    // ==============================
    // INTERNAL (optional)
    // ==============================
    aocSpeedTarget              : REAL;      // target line speed during AOC (m/min)
END_VAR

VAR CONSTANT
    // ==============================
    // LIFE CYCLE
    // ==============================
    STATUS_NO_CALL                  : WORD := 16#7000;
    STATUS_FB_FIRST_CALL            : WORD := 16#7001;

    // ==============================
    // AOC STATES
    // ==============================
    STATUS_CHECK_CONDITIONS         : WORD := 16#8000;
    STATUS_SAVE_DF_SPEED            : WORD := 16#8001;
    STATUS_REDUCE_DF_SPEED          : WORD := 16#8002;

    STATUS_ROTARY_SHEAR_CUT_X1      : WORD := 16#8003;
    STATUS_WAIT_ROTARY_SHEAR_CUT_X1 : WORD := 16#8103;

    STATUS_INCREASE_DRYEND_SPEED    : WORD := 16#8004;
    STATUS_CHANGE_SLT_ORDER         : WORD := 16#8005;
    STATUS_CHANGE_RK_SHEET_LENGTH   : WORD := 16#8006;
    STATUS_STK_DISCHARGE            : WORD := 16#8007;

    STATUS_AOC_FINISHED             : WORD := 16#8010;
END_VAR

// =================================================================================================
// CPNTeck - Automação ind.
// (c)Copyright 2022 All Rights Reserved
// -------------------------------------------------------------------------------------------------
// Purpose: Automatic Order Change (AOC) sequence controller.
// Steps (high-level):
//   1) Check material presence
//   2) Reduce double facer speed down to AOC speed
//   3) Execute single cut (rotary shear X1)
//   4) Switch reference to AOC ramp and clear dry-end/slitter
//   5) Update slitter parameters from nextOrder
//   6) Change rotary knife sheet length (delay / clearance window)
//   7) Discharge stacker
//   8) Finish and reset
//
// Notes (important):
// - TP/TON instances are called once per scan at the end of the FB.
// - Requests (reqTp*/reqTon*) are set inside the state machine.
// - This avoids conflicting multi-calls to the same FB instance.
// =================================================================================================


// =================================================================================================
// 1) EDGE HANDLING / DISABLE RESET
// =================================================================================================
rExecuteAOC := executeAOC AND NOT executeAOC_Old;
executeAOC_Old := executeAOC;

// Falling edge of enable => hard reset (safe state)
IF (NOT enable) AND enableOld THEN
    // ---- outputs ----
    error := FALSE;
    aocRunning := FALSE;
    aocTimeOut := FALSE;
    statusDisplay := 'Not running...';

    referenceSwitch := FALSE;
    doubleFacerSpeedUP := FALSE;
    doubleFacerSpeedDown := FALSE;

    rotaryShearCutX1 := FALSE;
    executePositioning := FALSE;
    topStackerDischarge := FALSE;
    bottomStackerDischarge := FALSE;

    rotaryKnifeSpeedRef := 0.0;
    slitterKnifeSpeedRef := 0.0;
    slitterScorerSpeedRef := 0.0;

    // ---- state ----
    stateMachine := STATUS_NO_CALL;

    // ---- reset requests ----
    reqTpRotaryShear := FALSE;
    reqTpExecutePositioning := FALSE;
    reqTpStackerTop := FALSE;
    reqTpStackerBottom := FALSE;

    reqTonSlitterDelay := FALSE;
    reqTonStackerDelay := FALSE;
    reqTonChangeSheetLength := FALSE;

    // ---- stop timeout ----
    tonAocTimeout.IN := FALSE;

    enableOld := enable;
    RETURN;
END_IF

// Rising edge of enable => initialize
IF enable AND (NOT enableOld) THEN
    stateMachine := STATUS_FB_FIRST_CALL;

    // Keep outputs in safe defaults
    error := FALSE;
    aocRunning := FALSE;
    aocTimeOut := FALSE;
    statusDisplay := 'Initialized';

    enableOld := enable;
    RETURN;
END_IF

// If not enabled, do nothing
IF NOT enable THEN
    enableOld := enable;
    RETURN;
END_IF

enableOld := enable;


// =================================================================================================
// 2) DEFAULTS EACH SCAN (avoid latching unwanted outputs)
// =================================================================================================
rotaryShearCutX1 := FALSE;
executePositioning := FALSE;
topStackerDischarge := FALSE;
bottomStackerDischarge := FALSE;

doubleFacerSpeedUP := FALSE;
doubleFacerSpeedDown := FALSE;

// Requests default OFF; states will enable them as needed
reqTpRotaryShear := FALSE;
reqTpExecutePositioning := FALSE;
reqTpStackerTop := FALSE;
reqTpStackerBottom := FALSE;

reqTonSlitterDelay := FALSE;
reqTonStackerDelay := FALSE;
reqTonChangeSheetLength := FALSE;


// =================================================================================================
// 3) TRIGGER AOC (rising edge)
// =================================================================================================
IF rExecuteAOC THEN
    aocTimeOut := FALSE;
    stateMachine := STATUS_CHECK_CONDITIONS;
END_IF


// =================================================================================================
// 4) STATE MACHINE
// =================================================================================================
CASE stateMachine OF

    STATUS_FB_FIRST_CALL:
        statusDisplay := 'FB first call';
        stateMachine := STATUS_NO_CALL;

    STATUS_NO_CALL:
        statusDisplay := 'Idle';
        aocRunning := FALSE;
        referenceSwitch := FALSE;
        tonAocTimeout.IN := FALSE;

    STATUS_CHECK_CONDITIONS:
        statusDisplay := 'Checking conditions';

        // Must have paper present everywhere to proceed
        IF (NOT measuringWheelPaperSensor)
           OR (NOT slitterPaperPresenceSensor)
           OR (NOT rotaryKnifePaperSensor) THEN

            // Not safe to run AOC, finish immediately
            stateMachine := STATUS_AOC_FINISHED;
        ELSE
            // Start timeout supervision
            tonAocTimeout.IN := TRUE;
            tonAocTimeout.PT := configuration.aocTimeout;

            stateMachine := STATUS_SAVE_DF_SPEED;
        END_IF


    STATUS_SAVE_DF_SPEED:
        statusDisplay := 'STATUS_SAVE_DF_SPEED';
        aocRunning := TRUE;

        // Compute AOC target speed (m/min)
        aocSpeedTarget := configuration.automaticOrderChangeSpeed * configuration.automaticOrderChangeSpeedMult;

        stateMachine := STATUS_REDUCE_DF_SPEED;


    STATUS_REDUCE_DF_SPEED:
        statusDisplay := 'STATUS_REDUCE_DF_SPEED';

        // While above AOC speed => pulse DF speed down
        IF lineSpeedMPM > configuration.automaticOrderChangeSpeed THEN
            doubleFacerSpeedDown := instGEN_PULSESpeedCtrl.Q;
        ELSE
            // Reached speed => go cut
            stateMachine := STATUS_ROTARY_SHEAR_CUT_X1;
        END_IF

        // Freeze ramp output to current speed (no AOC ramp yet)
        instFB_Gen_SRamp.X          := lineSpeedMPM;
        instFB_Gen_SRamp.LIMIT_LOW  := lineSpeedMPM;
        instFB_Gen_SRamp.LIMIT_HIGH := lineSpeedMPM;


    STATUS_ROTARY_SHEAR_CUT_X1:
        statusDisplay := 'Cutting web (X1)';
        // Generate a 1s pulse to the shear output
        reqTpRotaryShear := TRUE;
        stateMachine := STATUS_WAIT_ROTARY_SHEAR_CUT_X1;


    STATUS_WAIT_ROTARY_SHEAR_CUT_X1:
        statusDisplay := 'Waiting shear sensor';

        // Wait for confirmation sensor
        IF rotaryShearCutSensor THEN
            // Switch reference to AOC ramp
            referenceSwitch := TRUE;
            stateMachine := STATUS_INCREASE_DRYEND_SPEED;
        END_IF


    STATUS_INCREASE_DRYEND_SPEED:
        statusDisplay := 'Clearing dry-end / slitter';

        // Wait until measuring wheel area clears
        IF NOT measuringWheelPaperSensor THEN
            stateMachine := STATUS_CHANGE_SLT_ORDER;
        END_IF

        // Apply AOC speed ramp (raise limit high to target)
        instFB_Gen_SRamp.X          := aocSpeedTarget;
        instFB_Gen_SRamp.LIMIT_LOW  := lineSpeedMPM;     // don’t ramp below current
        instFB_Gen_SRamp.LIMIT_HIGH := aocSpeedTarget;


    STATUS_CHANGE_SLT_ORDER:
        statusDisplay := 'Changing slitter order (when clear)';

        // Copy only the parameters that need to switch during AOC
        currentOrder.fluteType     := nextOrder.fluteType;
        currentOrder.levelSelector := nextOrder.levelSelector;

        currentOrder.order1.sheetType     := nextOrder.order1.sheetType;
        currentOrder.order1.sheetQuantity := nextOrder.order1.sheetQuantity;
        currentOrder.order1.sheetM1       := nextOrder.order1.sheetM1;
        currentOrder.order1.sheetM2       := nextOrder.order1.sheetM2;
        currentOrder.order1.sheetM3       := nextOrder.order1.sheetM3;
        currentOrder.order1.sheetM4       := nextOrder.order1.sheetM4;
        currentOrder.order1.sheetM5       := nextOrder.order1.sheetM5;

        currentOrder.order2.sheetType     := nextOrder.order2.sheetType;
        currentOrder.order2.sheetQuantity := nextOrder.order2.sheetQuantity;
        currentOrder.order2.sheetM1       := nextOrder.order2.sheetM1;
        currentOrder.order2.sheetM2       := nextOrder.order2.sheetM2;
        currentOrder.order2.sheetM3       := nextOrder.order2.sheetM3;
        currentOrder.order2.sheetM4       := nextOrder.order2.sheetM4;
        currentOrder.order2.sheetM5       := nextOrder.order2.sheetM5;

        // Start delay only after slitter area becomes clear
        IF NOT slitterPaperPresenceSensor THEN
            reqTonSlitterDelay := TRUE;
            tonSlitterPresenceDelay.PT := configuration.slitterPaperPresenceDelay;
        END_IF

        IF tonSlitterPresenceDelay.Q THEN
            // Pulse executePositioning
            reqTpExecutePositioning := TRUE;

            // stop delay timer (will reset by IN=FALSE)
            reqTonSlitterDelay := FALSE;

            stateMachine := STATUS_CHANGE_RK_SHEET_LENGTH;
        END_IF


    STATUS_CHANGE_RK_SHEET_LENGTH:
        statusDisplay := 'Changing rotary knife sheet length';

        // Allow a clearance window for RK sheet length change (time-based + sensor-based)
        reqTonChangeSheetLength := TRUE;
        tonChangeSheetLength.PT := configuration.changeSheetLengthTime;

        // When RK is clear OR timer elapsed => proceed
        IF (NOT rotaryKnifePaperSensor) OR tonChangeSheetLength.Q THEN
            reqTonChangeSheetLength := FALSE;
			currentOrder.changeOrderRequest := TRUE;
            stateMachine := STATUS_STK_DISCHARGE;
        END_IF


    STATUS_STK_DISCHARGE:
        statusDisplay := 'Discharging stacker';

        // Delay before discharge
        reqTonStackerDelay := TRUE;
        tonStackerDischargeDelay.PT := configuration.stackerDischargeDelay;

        IF tonStackerDischargeDelay.Q THEN
            // Pulse discharge commands
            reqTpStackerTop := TRUE;
            reqTpStackerBottom := TRUE;

            // Once pulses are done, finish
            // (TP outputs will be active for PT time; we can finish immediately or wait—here we finish)
            stateMachine := STATUS_AOC_FINISHED;
        END_IF


    STATUS_AOC_FINISHED:
        statusDisplay := 'AOC Finished';

        aocRunning := FALSE;
        referenceSwitch := FALSE;
        doubleFacerSpeedUP := FALSE;
        doubleFacerSpeedDown := FALSE;

        // Stop timeout monitoring
        tonAocTimeout.IN := FALSE;

        // Return to idle
        stateMachine := STATUS_NO_CALL;

END_CASE


// =================================================================================================
// 5) GLOBAL FUNCTION BLOCK CALLS (call once per scan)
// =================================================================================================

// Pulse generator for DF speed up/down buttons
instGEN_PULSESpeedCtrl(
    ENQ := TRUE,
    PTH := configuration.speedControlPulseONTime,
    PTL := configuration.speedControlPulseOFFTime
);

// Ramp block (driven by instFB_Gen_SRamp.X and limits set in states)
instFB_Gen_SRamp(
    A_UP    := configuration.rampUpTimeSec,
    A_DN    := configuration.rampDownTimeSec,
    VU_MAX  := 1000.0,
    VD_MAX  := -1000.0,
    Y       => lineSpeedMPMRamp
);

// Timers
tonSlitterPresenceDelay(IN := reqTonSlitterDelay);
tonStackerDischargeDelay(IN := reqTonStackerDelay);
tonChangeSheetLength(IN := reqTonChangeSheetLength);

tonAocTimeout(IN := tonAocTimeout.IN, PT := configuration.aocTimeout);

// Pulses
tpRotaryShear(IN := reqTpRotaryShear, PT := T#1S, Q => rotaryShearCutX1);
tpExecutePositioning(IN := reqTpExecutePositioning, PT := T#1S, Q => executePositioning);
tpStackerTop(IN := reqTpStackerTop, PT := T#1S, Q => topStackerDischarge);
tpStackerBottom(IN := reqTpStackerBottom, PT := T#1S, Q => bottomStackerDischarge);


// =================================================================================================
// 6) REFERENCES (derived from ramp output)
// =================================================================================================
rotaryKnifeSpeedRef   := lineSpeedMPMRamp * configuration.rotaryKnifeSpeedMult;
slitterKnifeSpeedRef  := lineSpeedMPMRamp * configuration.slitterSpeedMult;
slitterScorerSpeedRef := lineSpeedMPMRamp * configuration.slitterSpeedMult;


// =================================================================================================
// 7) TIMEOUT HANDLING
// =================================================================================================
IF tonAocTimeout.Q THEN
    tonAocTimeout.IN := FALSE;
    aocTimeOut := TRUE;
    stateMachine := STATUS_AOC_FINISHED;
END_IF

END_FUNCTION_BLOCK

// ---- Library/Machine/Rotary knife/Function Block/FB_RotaryKnife_1.TcPOU
FUNCTION_BLOCK FB_RotaryKnife_1




VAR_OUTPUT
    //────────────────────────────────────────────
    // GENERAL / ALARMS (COMMON)
    //────────────────────────────────────────────
    alarmActive                     : BOOL;  // Global alarm active / Alarme geral ativo

    //────────────────────────────────────────────
    // UPPER LEVEL — ENABLE / RUN COMMANDS
    //────────────────────────────────────────────
    upperLevelEnable                : BOOL;  // Upper level enable / Habilita nível superior
    upperLevelInFeedRun             : BOOL;  // Upper infeed run / Partida infeed superior
    upperLevelOutFeedRun            : BOOL;  // Upper outfeed run / Partida outfeed superior
    upperLevelSlave1Run             : BOOL;  // Upper slave1 run / Partida slave1 superior
    upperLevelSlave2Run             : BOOL;  // Upper slave2 run / Partida slave2 superior

    //────────────────────────────────────────────
    // UPPER LEVEL — MOTION / CUT / HOME COMMANDS
    //────────────────────────────────────────────
    upperLevelJogFw                 : BOOL;  // Upper jog forward / JOG avanço superior
    upperLevelJogRev                : BOOL;  // Upper jog reverse / JOG reverso superior
    upperLevelCut                   : BOOL;  // Upper cut command output / Saída corte superior
    upperLevelHome                  : BOOL;  // Upper home command output / Saída home superior
    upperLevelHomeSensorPulse       : BOOL;  // Upper home sensor pulse / Pulso sensor home superior

    //────────────────────────────────────────────
    // UPPER LEVEL — RESET STATUS
    //────────────────────────────────────────────
    upperLevelReset                 : BOOL;  // Upper reset active / Reset superior ativo

    //────────────────────────────────────────────
    // UPPER LEVEL — SPEED REFERENCES
    //────────────────────────────────────────────
    upperLevelInFeedDriveRef        : REAL;  // Upper infeed speed reference / Referência velocidade infeed superior
    upperLevelOutFeedDriveRef       : REAL;  // Upper outfeed speed reference / Referência velocidade outfeed superior

    //────────────────────────────────────────────
    // UPPER LEVEL — ENCODER SELECTION OUTPUT
    //────────────────────────────────────────────
    upperLevelEncoderSwitch         : BOOL;  // Upper encoder select (to drive/IO) / Seletor encoder superior

    //────────────────────────────────────────────
    // LOWER LEVEL — ENABLE / RUN COMMANDS (CREATED)
    //────────────────────────────────────────────
    lowerLevelEnable                : BOOL;  // Lower level enable / Habilita nível inferior
    lowerLevelInFeedRun             : BOOL;  // Lower infeed run / Partida infeed inferior
    lowerLevelOutFeedRun            : BOOL;  // Lower outfeed run / Partida outfeed inferior
    lowerLevelSlave1Run             : BOOL;  // Lower slave1 run / Partida slave1 inferior
    lowerLevelSlave2Run             : BOOL;  // Lower slave2 run / Partida slave2 inferior

    //────────────────────────────────────────────
    // LOWER LEVEL — MOTION / CUT / HOME COMMANDS (CREATED)
    //────────────────────────────────────────────
    lowerLevelJogFw                 : BOOL;  // Lower jog forward / JOG avanço inferior
    lowerLevelJogRev                : BOOL;  // Lower jog reverse / JOG reverso inferior
    lowerLevelCut                   : BOOL;  // Lower cut command output / Saída corte inferior
    lowerLevelHome                  : BOOL;  // Lower home command output / Saída home inferior
    lowerLevelHomeSensorPulse       : BOOL;  // Lower home sensor pulse / Pulso sensor home inferior

    //────────────────────────────────────────────
    // LOWER LEVEL — RESET STATUS (CREATED)
    //────────────────────────────────────────────
    lowerLevelReset                 : BOOL;  // Lower reset active / Reset inferior ativo

    //────────────────────────────────────────────
    // LOWER LEVEL — SPEED REFERENCES (CREATED)
    //────────────────────────────────────────────
    lowerLevelInFeedDriveRef        : REAL;  // Lower infeed speed reference / Referência velocidade infeed inferior
    lowerLevelOutFeedDriveRef       : REAL;  // Lower outfeed speed reference / Referência velocidade outfeed inferior

    //────────────────────────────────────────────
    // LOWER LEVEL — ENCODER SELECTION OUTPUT (CREATED)
    //────────────────────────────────────────────
    lowerLevelEncoderSwitch         : BOOL;  // Lower encoder select (to drive/IO) / Seletor encoder inferior

    //────────────────────────────────────────────
    // HMI STATUS (COMMON)
    //────────────────────────────────────────────
    hmiStatus                       : hmiStatus_TypeStruct; // HMI status structure / Estrutura status HMI
END_VAR
VAR
    //────────────────────────────────────────────
    // UPPER LEVEL — INTERNAL SEQUENCE / STATE
    //────────────────────────────────────────────
    upperLevelStep                 : INT := 0;      // Sequence step for upper level

    //────────────────────────────────────────────
    // UPPER LEVEL — INTERNAL AGGREGATIONS / FLAGS
    //────────────────────────────────────────────
    upperLevelAllDrivesOK          : BOOL := FALSE; // Aggregated drive OK status

    //────────────────────────────────────────────
    // UPPER LEVEL — EDGE DETECTORS
    //────────────────────────────────────────────
    upperLevelRtEnable             : R_TRIG;        // Rising edge for Power ON command
    upperLevelRtPowerOff           : R_TRIG;        // Rising edge for Power OFF command

    //────────────────────────────────────────────
    // UPPER LEVEL — TIMERS
    //────────────────────────────────────────────
    upperLevelTimerReset           : TON;           // 2s reset pulse timer
    upperLevelTimerPulse           : TON;           // General wait/pulse timer used in step 20
    upperLevelTimerWait            : TON;           // Reserved (used in safety reset section)
    upperLevelTimerClear           : TON;           // Reserved (used in safety reset section)

    //────────────────────────────────────────────
    // LOWER LEVEL — INTERNAL SEQUENCE / STATE (CREATED)
    //────────────────────────────────────────────
    lowerLevelStep                 : INT := 0;      // Sequence step for lower level

    //────────────────────────────────────────────
    // LOWER LEVEL — INTERNAL AGGREGATIONS / FLAGS (CREATED)
    //────────────────────────────────────────────
    lowerLevelAllDrivesOK          : BOOL := FALSE; // Aggregated drive OK status

    //────────────────────────────────────────────
    // LOWER LEVEL — EDGE DETECTORS (CREATED)
    //────────────────────────────────────────────
    lowerLevelRtEnable             : R_TRIG;        // Rising edge for Power ON command
    lowerLevelRtPowerOff           : R_TRIG;        // Rising edge for Power OFF command

    //────────────────────────────────────────────
    // LOWER LEVEL — TIMERS (CREATED)
    //────────────────────────────────────────────
    lowerLevelTimerReset           : TON;           // 2s reset pulse timer
    lowerLevelTimerPulse           : TON;           // General wait/pulse timer used in step 20
    lowerLevelTimerWait            : TON;           // Reserved (used in safety reset section)
    lowerLevelTimerClear           : TON;           // Reserved (used in safety reset section)

    //────────────────────────────────────────────
    // MODBUS TCP — FUNCTION BLOCKS / GLOBAL STATE
    //────────────────────────────────────────────
    instFB_MBReadRegs              : FB_MBReadRegs;   // Modbus TCP read registers FB
    instFB_MBWriteRegs             : FB_MBWriteRegs;  // Modbus TCP write registers FB
    modbusTCPStep                  : INT;             // Modbus TCP state machine step

    //────────────────────────────────────────────
    // MODBUS TCP — UPPER LEVEL DATA
    //────────────────────────────────────────────
    upperLevelStatusWord1          : INT;
    upperLevelStatusWord2          : INT;
    upperLevelModbusDword          : DWORD;
    upperLevelWriteMenu2029        : DWORD;
    upperLevelLineSpeed            : WORD;
	upperLevelStatusW1				: rotaryKnifeStatusWord1_TypeStruct;
	upperLevelStatusW2				: rotaryKnifeStatusWord2_TypeStruct;		

    //────────────────────────────────────────────
    // MODBUS TCP — LOWER LEVEL DATA
    //────────────────────────────────────────────
    lowerLevelStatusWord1          : INT;
    lowerLevelStatusWord2          : INT;
    lowerLevelModbusDword          : DWORD;
    lowerLevelWriteMenu2029        : DWORD;
    lowerLevelLineSpeed            : WORD;

	lowerLevelStatusW1				: rotaryKnifeStatusWord1_TypeStruct;
	lowerLevelStatusW2				: rotaryKnifeStatusWord2_TypeStruct;	
	
	
END_VAR

VAR PERSISTENT
	
	lowerLevelTotalOfCutsAccumulator : DINT;
	upperLevelTotalOfCutsAccumulator : DINT;


END_VAR

VAR_IN_OUT

	currentOrder	: Order_TypeStruct;

END_VAR

_00_ModbusTCP();
_01_UpperLevelControl();
_02_LowerLevelControl();

METHOD _00_ModbusTCP
VAR_INPUT
END_VAR
CASE modbusTCPStep OF
	
		(*________________________________________________________________*)
		00:(*Read lower level line speed*)
	
		instFB_MBReadRegs(
		sIPAddr:= '192.168.100.11', 
		nTCPPort:= 502, 
		nUnitID:= 1, 
		nQuantity:= 1, 
		nMBAddr:= 16#711, (*Menu 18.10*)
		cbLength:= SIZEOF(lowerLevelLineSpeed),  
		pDestAddr:= ADR(lowerLevelLineSpeed),  
		bExecute:= TRUE, 
		tTimeout:= T#500MS,  
		bBusy=> , 
		bError=> , 
		nErrId=> , 
		cbRead=> );
		
	
		IF NOT instFB_MBReadRegs.bBusy THEN
			instFB_MBReadRegs(bExecute:=FALSE);
			modbusTCPStep:=modbusTCPStep + 1;	(*Index*)
		END_IF
		
		
		(*________________________________________________________________*)		
		01:(*Read rotary knife status word1*)
	
		instFB_MBReadRegs(
		sIPAddr:= '192.168.100.11', 
		nTCPPort:= 502, 
		nUnitID:= 1, 
		nQuantity:= 1, 
		nMBAddr:= 16#774, //Parameter #19.09 - 1 = > HEX
		cbLength:= SIZEOF(upperLevelStatusWord1),  
		pDestAddr:= ADR(upperLevelStatusWord1),  
		bExecute:= TRUE,  
		tTimeout:= T#500MS,  
		bBusy=> , 
		bError=> , 
		nErrId=> , 
		cbRead=> );
		
		IF NOT instFB_MBReadRegs.bBusy THEN
			instFB_MBReadRegs(bExecute:=FALSE);
			modbusTCPStep:=modbusTCPStep + 1;	(*Index*)			
		END_IF	
		
		
		(*________________________________________________________________*)		
		02:(*Read rotary knife status word1*)
	
		instFB_MBReadRegs(
		sIPAddr:= '192.168.100.11', 
		nTCPPort:= 502, 
		nUnitID:= 1, 
		nQuantity:= 1, 
		nMBAddr:= 16#775, //Parameter #19.10 - 1 = > HEX
		cbLength:= SIZEOF(upperLevelStatusWord2),  
		pDestAddr:= ADR(upperLevelStatusWord2),  
		bExecute:= TRUE,  
		tTimeout:= T#500MS,  
		bBusy=> , 
		bError=> , 
		nErrId=> , 
		cbRead=> );
		
		IF NOT instFB_MBReadRegs.bBusy THEN
			instFB_MBReadRegs(bExecute:=FALSE);
			modbusTCPStep:=modbusTCPStep + 1;	(*Index*)

		END_IF			





		(*________________________________________________________________*)
		03:(*Read lower level line speed*)
	
		instFB_MBReadRegs(
		sIPAddr:= '192.168.100.12', 
		nTCPPort:= 502, 
		nUnitID:= 1, 
		nQuantity:= 1, 
		nMBAddr:= 16#711, (*Menu 18.10*)
		cbLength:= SIZEOF(lowerLevelLineSpeed),  
		pDestAddr:= ADR(lowerLevelLineSpeed),  
		bExecute:= TRUE, 
		tTimeout:= T#500MS,  
		bBusy=> , 
		bError=> , 
		nErrId=> , 
		cbRead=> );
		
	
		IF NOT instFB_MBReadRegs.bBusy THEN
			instFB_MBReadRegs(bExecute:=FALSE);
			modbusTCPStep:=modbusTCPStep + 1;	(*Index*)
		END_IF
		
		
		(*________________________________________________________________*)		
		04:(*Read rotary knife status word1*)
	
		instFB_MBReadRegs(
		sIPAddr:= '192.168.100.12', 
		nTCPPort:= 502, 
		nUnitID:= 1, 
		nQuantity:= 1, 
		nMBAddr:= 16#774, //Parameter #19.09 - 1 = > HEX
		cbLength:= SIZEOF(lowerLevelStatusWord1),  
		pDestAddr:= ADR(lowerLevelStatusWord1),  
		bExecute:= TRUE,  
		tTimeout:= T#500MS,  
		bBusy=> , 
		bError=> , 
		nErrId=> , 
		cbRead=> );
		
		
		IF NOT instFB_MBReadRegs.bBusy THEN
			instFB_MBReadRegs(bExecute:=FALSE);
			modbusTCPStep:=modbusTCPStep + 1;	(*Index*)			
		END_IF	
		
		(*________________________________________________________________*)		
		05:(*Read rotary knife status word1*)
	
		instFB_MBReadRegs(
		sIPAddr:= '192.168.100.12', 
		nTCPPort:= 502, 
		nUnitID:= 1, 
		nQuantity:= 1, 
		nMBAddr:= 16#775, //Parameter #19.10 - 1 = > HEX
		cbLength:= SIZEOF(lowerLevelStatusWord2),  
		pDestAddr:= ADR(lowerLevelStatusWord2),  
		bExecute:= TRUE,  
		tTimeout:= T#500MS,  
		bBusy=> , 
		bError=> , 
		nErrId=> , 
		cbRead=> );
		
		IF NOT instFB_MBReadRegs.bBusy THEN
			instFB_MBReadRegs(bExecute:=FALSE);
			modbusTCPStep:=modbusTCPStep + 1;	(*Index*)

		END_IF	
		
		
		
	(*________________________________________________________________*)	
		6:(*Write lower level sheet lenght*)	
	
		
		IF NOT currentOrder.invertOrderLevel THEN
			
			upperLevelModbusDword := (INT_TO_DWORD(currentOrder.order1.sheetLength) * 1000);
	
		ELSE
			
			upperLevelModbusDword := (INT_TO_DWORD(currentOrder.order2.sheetLength) * 1000);			
		
		END_IF
					
		upperLevelWriteMenu2029 := SHR(upperLevelModbusDword,16) OR SHL(upperLevelModbusDword,16);
		
		//Write menu 20.29 - MBAddres: 16#47EC (18412dec)
		instFB_MBWriteRegs(
		sIPAddr:= '192.168.100.11', //Modbus gateway IP Addres
		nTCPPort:= 502, //Modbus gateway port
		nUnitID:= 1, //Drive addres subnode
		nQuantity:= 2, //Number of words
		nMBAddr:= 16#47EC, 
		cbLength:= SIZEOF(upperLevelWriteMenu2029), 
		pSrcAddr:= ADR(upperLevelWriteMenu2029), 
		bExecute:= TRUE, 
		tTimeout:= T#1000MS, 
		bBusy=> , 
		bError=> , 
		nErrId=> );
		
		IF NOT instFB_MBWriteRegs.bBusy THEN
			instFB_MBWriteRegs(bExecute:=FALSE);
			modbusTCPStep:=modbusTCPStep + 1;	(*Index*)

		END_IF			

		
		
		7:(*Write lower level sheet lenght*)	
	
		
		IF NOT currentOrder.invertOrderLevel THEN
			
			lowerLevelModbusDword := (INT_TO_DWORD(currentOrder.order2.sheetLength) * 1000);
	
		ELSE
			
			lowerLevelModbusDword := (INT_TO_DWORD(currentOrder.order1.sheetLength) * 1000);			
		
		END_IF
					
		lowerLevelWriteMenu2029 := SHR(lowerLevelModbusDword,16) OR SHL(lowerLevelModbusDword,16);
		
		//Write menu 20.29 - MBAddres: 16#47EC (18412dec)
		instFB_MBWriteRegs(
		sIPAddr:= '192.168.100.12', //Modbus gateway IP Addres
		nTCPPort:= 502, //Modbus gateway port
		nUnitID:= 1, //Drive addres subnode
		nQuantity:= 2, //Number of words
		nMBAddr:= 16#47EC, 
		cbLength:= SIZEOF(lowerLevelWriteMenu2029), 
		pSrcAddr:= ADR(lowerLevelWriteMenu2029), 
		bExecute:= TRUE, 
		tTimeout:= T#1000MS, 
		bBusy=> , 
		bError=> , 
		nErrId=> );
		
		IF NOT instFB_MBWriteRegs.bBusy THEN
			instFB_MBWriteRegs(bExecute:=FALSE);
			modbusTCPStep:=0;	(*Index*)

		END_IF				
	
END_CASE		



//==============================================================
// STATUS WORD 1 — BIT TO BOOL MAPPING (Upper + Lower)
//==============================================================

//-----------------------------
// Upper Level — Status Word 1
//-----------------------------
upperLevelStatusW1.knifeAtHomeParkPos1              := upperLevelStatusWord1.00;
upperLevelStatusW1.homingInProgress                 := upperLevelStatusWord1.01;
upperLevelStatusW1.homingComplete                   := upperLevelStatusWord1.02;
upperLevelStatusW1.knifeInspectionMotionInProgress  := upperLevelStatusWord1.03;
upperLevelStatusW1.knifeInspectionMotionComplete    := upperLevelStatusWord1.04;
upperLevelStatusW1.returnHomeMotionInProgress       := upperLevelStatusWord1.05;
upperLevelStatusW1.returnHomeMotionComplete         := upperLevelStatusWord1.06;
upperLevelStatusW1.jogForwardInProgress             := upperLevelStatusWord1.07;
upperLevelStatusW1.jogReverseInProgress             := upperLevelStatusWord1.08;
upperLevelStatusW1.knifeGearingOut                  := upperLevelStatusWord1.09;
upperLevelStatusW1.knifeRunningEngaged              := upperLevelStatusWord1.10;
upperLevelStatusW1.knifeStoppedDisengaged           := upperLevelStatusWord1.11;
upperLevelStatusW1.maxLineSpeedLimitCalculated      := upperLevelStatusWord1.12;
upperLevelStatusW1.batchMaxLineSpeedCalcInProgress  := upperLevelStatusWord1.13;
upperLevelStatusW1.batchMaxLineSpeedCalculated      := upperLevelStatusWord1.14;
upperLevelStatusW1.watchdogClockOut                 := upperLevelStatusWord1.15;

//-----------------------------
// Lower Level — Status Word 1
//-----------------------------
lowerLevelStatusW1.knifeAtHomeParkPos1              := lowerLevelStatusWord1.00;
lowerLevelStatusW1.homingInProgress                 := lowerLevelStatusWord1.01;
lowerLevelStatusW1.homingComplete                   := lowerLevelStatusWord1.02;
lowerLevelStatusW1.knifeInspectionMotionInProgress  := lowerLevelStatusWord1.03;
lowerLevelStatusW1.knifeInspectionMotionComplete    := lowerLevelStatusWord1.04;
lowerLevelStatusW1.returnHomeMotionInProgress       := lowerLevelStatusWord1.05;
lowerLevelStatusW1.returnHomeMotionComplete         := lowerLevelStatusWord1.06;
lowerLevelStatusW1.jogForwardInProgress             := lowerLevelStatusWord1.07;
lowerLevelStatusW1.jogReverseInProgress             := lowerLevelStatusWord1.08;
lowerLevelStatusW1.knifeGearingOut                  := lowerLevelStatusWord1.09;
lowerLevelStatusW1.knifeRunningEngaged              := lowerLevelStatusWord1.10;
lowerLevelStatusW1.knifeStoppedDisengaged           := lowerLevelStatusWord1.11;
lowerLevelStatusW1.maxLineSpeedLimitCalculated      := lowerLevelStatusWord1.12;
lowerLevelStatusW1.batchMaxLineSpeedCalcInProgress  := lowerLevelStatusWord1.13;
lowerLevelStatusW1.batchMaxLineSpeedCalculated      := lowerLevelStatusWord1.14;
lowerLevelStatusW1.watchdogClockOut                 := lowerLevelStatusWord1.15;

//==============================================================
// STATUS WORD 2 — BIT TO BOOL MAPPING (Upper + Lower)
//==============================================================

//-----------------------------
// Upper Level — Status Word 2
//-----------------------------
upperLevelStatusW2.batchSingleShotStopInProgress := upperLevelStatusWord2.00;
upperLevelStatusW2.registrationMarkMissed        := upperLevelStatusWord2.01;
upperLevelStatusW2.registrationWindowOpen        := upperLevelStatusWord2.02;
upperLevelStatusW2.registrationMarkAccepted      := upperLevelStatusWord2.03;
upperLevelStatusW2.onLastBatch                   := upperLevelStatusWord2.04;
upperLevelStatusW2.onLastCutOfLastBatch          := upperLevelStatusWord2.05;
upperLevelStatusW2.pls1Output                    := upperLevelStatusWord2.06;
upperLevelStatusW2.pls2Output                    := upperLevelStatusWord2.07;
upperLevelStatusW2.referenceEnabled              := upperLevelStatusWord2.08;
upperLevelStatusW2.driveHealthy                  := upperLevelStatusWord2.09;
upperLevelStatusW2.reserved10                    := upperLevelStatusWord2.10;
upperLevelStatusW2.reserved11                    := upperLevelStatusWord2.11;
upperLevelStatusW2.userDefinedStatusBit12        := upperLevelStatusWord2.12;
upperLevelStatusW2.userDefinedStatusBit13        := upperLevelStatusWord2.13;
upperLevelStatusW2.userDefinedStatusBit14        := upperLevelStatusWord2.14;
upperLevelStatusW2.userDefinedStatusBit15        := upperLevelStatusWord2.15;

//-----------------------------
// Lower Level — Status Word 2
//-----------------------------
lowerLevelStatusW2.batchSingleShotStopInProgress := lowerLevelStatusWord2.00;
lowerLevelStatusW2.registrationMarkMissed        := lowerLevelStatusWord2.01;
lowerLevelStatusW2.registrationWindowOpen        := lowerLevelStatusWord2.02;
lowerLevelStatusW2.registrationMarkAccepted      := lowerLevelStatusWord2.03;
lowerLevelStatusW2.onLastBatch                   := lowerLevelStatusWord2.04;
lowerLevelStatusW2.onLastCutOfLastBatch          := lowerLevelStatusWord2.05;
lowerLevelStatusW2.pls1Output                    := lowerLevelStatusWord2.06;
lowerLevelStatusW2.pls2Output                    := lowerLevelStatusWord2.07;
lowerLevelStatusW2.referenceEnabled              := lowerLevelStatusWord2.08;
lowerLevelStatusW2.driveHealthy                  := lowerLevelStatusWord2.09;
lowerLevelStatusW2.reserved10                    := lowerLevelStatusWord2.10;
lowerLevelStatusW2.reserved11                    := lowerLevelStatusWord2.11;
lowerLevelStatusW2.userDefinedStatusBit12        := lowerLevelStatusWord2.12;
lowerLevelStatusW2.userDefinedStatusBit13        := lowerLevelStatusWord2.13;
lowerLevelStatusW2.userDefinedStatusBit14        := lowerLevelStatusWord2.14;
lowerLevelStatusW2.userDefinedStatusBit15        := lowerLevelStatusWord2.15;
END_METHOD

METHOD _01_UpperLevelControl
VAR_INPUT
END_VAR
(*
======================================================================
UPPER LEVEL — Rotary Knife Control (Upper Knife)
======================================================================
Concept:
- Power ON command starts a simple sequence:
  0  = OFF / Idle
  10 = Enable drives + follow line speed
  20 = Send HOME command for 1s
  21 = Wait for HomingComplete status before running infeed/outfeed
  40 = Normal operation (cut enabled when command + paper present)

Rule:
- When the upper level is powered ON, infeed/outfeed speed references
  must follow lineSpeedMPM.
======================================================================
*)

//==============================================================
// 1) RESET PULSE (2s) + EDGE DETECTION
//==============================================================
upperLevelTimerReset(IN := resetCmd, PT := T#2S);
upperLevelReset := upperLevelTimerReset.Q;

upperLevelRtEnable(CLK := upperLevelPowerONCmd);
upperLevelRtPowerOff(CLK := upperLevelPowerOFFCmd);

//==============================================================
// 2) DRIVE/SAFETY STATUS (AGGREGATION)
//==============================================================
upperLevelAllDrivesOK := upperLevelInfeedDrvOK  AND
                         upperLevelOutfeedDrvOK AND
                         upperLevelMainDrvOK    AND
                         upperLevelSlave1DrvOK  AND
                         upperLevelSlave2DrvOK;

upperLevelHomeSensorPulse := upperLevelHomeSensor;

//==============================================================
// 3) START SEQUENCE CONDITION
//==============================================================
// Start only if:
// - Rising edge on Power ON
// - Sequence is idle
// - Safety chain OK
// - All drives OK
// - No reset pulse active
IF upperLevelRtEnable.Q
   AND (upperLevelStep = 0)
   AND safetyFeedback
   AND upperLevelAllDrivesOK
   AND NOT upperLevelReset THEN

    upperLevelStep := 10;
END_IF

//==============================================================
// 4) SEQUENCE STATE MACHINE
//==============================================================
CASE upperLevelStep OF

    //==========================================================
    // 0 — OFF / IDLE
    //==========================================================
    0:
        // Commands OFF
        upperLevelEnable      := FALSE;
        upperLevelSlave1Run   := FALSE;
        upperLevelSlave2Run   := FALSE;
        upperLevelInFeedRun   := FALSE;
        upperLevelOutFeedRun  := FALSE;

        // Motion / actions OFF
        upperLevelJogFw       := FALSE;
        upperLevelJogRev      := FALSE;
        upperLevelHome        := FALSE;
        upperLevelCut         := FALSE;

        // References = 0
        upperLevelInFeedDriveRef  := 0.0;
        upperLevelOutFeedDriveRef := 0.0;

    //==========================================================
    // 10 — ENABLE DRIVES + FOLLOW LINE SPEED
    //==========================================================
    10:
        upperLevelEnable      := TRUE;
        upperLevelSlave1Run   := TRUE;
        upperLevelSlave2Run   := TRUE;

        // Follow line speed immediately when powered ON
        upperLevelInFeedDriveRef  := lineSpeedMPM;
        upperLevelOutFeedDriveRef := lineSpeedMPM;

        // Next step: issue homing pulse
        upperLevelStep := 20;

    //==========================================================
    // 20 — HOME COMMAND PULSE (1s)
    //==========================================================
    20:
        // Command home for 1 second
        upperLevelHome := TRUE;

        upperLevelTimerPulse(IN := TRUE, PT := T#1S);
        IF upperLevelTimerPulse.Q THEN
            upperLevelHome := FALSE;
            upperLevelTimerPulse(IN := FALSE);
            upperLevelStep := 21;
        END_IF

    //==========================================================
    // 21 — WAIT HOMING COMPLETE
    //==========================================================
    21:

        // Start infeed/outfeed only after homing is complete
        IF upperLevelStatusW1.homingComplete THEN
            upperLevelInFeedRun  := TRUE;
            upperLevelOutFeedRun := TRUE;
            upperLevelStep := 40;
        END_IF

    //==========================================================
    // 40 — NORMAL OPERATION
    //==========================================================
    40:
        // Track line speed continuously
        upperLevelInFeedDriveRef  := lineSpeedMPM;
        upperLevelOutFeedDriveRef := lineSpeedMPM;

        // Enable cut only when commanded and paper present
        upperLevelCut := (upperLevelCutCmd AND upperLevelPaperSensor);

END_CASE

//==============================================================
// 5) GLOBAL INTERLOCK — IMMEDIATE STOP
//==============================================================
// Immediate stop on any of these conditions:
// - Safety chain not OK
// - Any drive not OK
// - Power OFF command rising edge
IF (NOT safetyFeedback) OR (NOT upperLevelAllDrivesOK) OR upperLevelRtPowerOff.Q THEN

    upperLevelStep := 0;

    upperLevelEnable      := FALSE;
    upperLevelSlave1Run   := FALSE;
    upperLevelSlave2Run   := FALSE;
    upperLevelInFeedRun   := FALSE;
    upperLevelOutFeedRun  := FALSE;

    upperLevelJogFw       := FALSE;
    upperLevelJogRev      := FALSE;
    upperLevelHome        := FALSE;
    upperLevelCut         := FALSE;

    upperLevelInFeedDriveRef  := 0.0;
    upperLevelOutFeedDriveRef := 0.0;

    // Reset internal timers for a clean restart
    upperLevelTimerWait(IN := FALSE);
    upperLevelTimerPulse(IN := FALSE);
    upperLevelTimerClear(IN := FALSE);
    upperLevelTimerReset(IN := FALSE);
END_IF
END_METHOD

METHOD _02_LowerLevelControl
VAR_INPUT
END_VAR
(*
======================================================================
LOWER LEVEL — Rotary Knife Control (Lower Knife)
======================================================================
Concept:
- Power ON command starts a simple sequence:
  0  = OFF / Idle
  10 = Enable drives + follow line speed
  20 = Send HOME command for 1s
  21 = Wait for HomingComplete status before running infeed/outfeed
  40 = Normal operation (cut enabled when command + paper present)

Rule:
- When the lower level is powered ON, infeed/outfeed speed references
  must follow lineSpeedMPM.
======================================================================
*)

//==============================================================
// 1) RESET PULSE (2s) + EDGE DETECTION
//==============================================================
lowerLevelTimerReset(IN := resetCmd, PT := T#2S);
lowerLevelReset := lowerLevelTimerReset.Q;

lowerLevelRtEnable(CLK := lowerLevelPowerONCmd);
lowerLevelRtPowerOff(CLK := lowerLevelPowerOFFCmd);

//==============================================================
// 2) DRIVE/SAFETY STATUS (AGGREGATION)
//==============================================================
lowerLevelAllDrivesOK := lowerLevelInfeedDrvOK  AND
                         lowerLevelOutfeedDrvOK AND
                         lowerLevelMainDrvOK    AND
                         lowerLevelSlave1DrvOK  AND
                         lowerLevelSlave2DrvOK;

lowerLevelHomeSensorPulse := lowerLevelHomeSensor;

//==============================================================
// 3) START SEQUENCE CONDITION
//==============================================================
// Start only if:
// - Rising edge on Power ON
// - Sequence is idle
// - Safety chain OK
// - All drives OK
// - No reset pulse active
IF lowerLevelRtEnable.Q
   AND (lowerLevelStep = 0)
   AND safetyFeedback
   AND lowerLevelAllDrivesOK
   AND NOT lowerLevelReset THEN

    lowerLevelStep := 10;
END_IF

//==============================================================
// 4) SEQUENCE STATE MACHINE
//==============================================================
CASE lowerLevelStep OF

    //==========================================================
    // 0 — OFF / IDLE
    //==========================================================
    0:
        // Commands OFF
        lowerLevelEnable      := FALSE;
        lowerLevelSlave1Run   := FALSE;
        lowerLevelSlave2Run   := FALSE;
        lowerLevelInFeedRun   := FALSE;
        lowerLevelOutFeedRun  := FALSE;

        // Motion / actions OFF
        lowerLevelJogFw       := FALSE;
        lowerLevelJogRev      := FALSE;
        lowerLevelHome        := FALSE;
        lowerLevelCut         := FALSE;

        // References = 0
        lowerLevelInFeedDriveRef  := 0.0;
        lowerLevelOutFeedDriveRef := 0.0;

    //==========================================================
    // 10 — ENABLE DRIVES + FOLLOW LINE SPEED
    //==========================================================
    10:
        lowerLevelEnable      := TRUE;
        lowerLevelSlave1Run   := TRUE;
        lowerLevelSlave2Run   := TRUE;

        // Follow line speed immediately when powered ON
        lowerLevelInFeedDriveRef  := lineSpeedMPM;
        lowerLevelOutFeedDriveRef := lineSpeedMPM;

        // Next step: issue homing pulse
        lowerLevelStep := 20;

    //==========================================================
    // 20 — HOME COMMAND PULSE (1s)
    //==========================================================
    20:
        // Command home for 1 second
        lowerLevelHome := TRUE;

        lowerLevelTimerPulse(IN := TRUE, PT := T#1S);
        IF lowerLevelTimerPulse.Q THEN
            lowerLevelHome := FALSE;
            lowerLevelTimerPulse(IN := FALSE);
            lowerLevelStep := 21;
        END_IF

    //==========================================================
    // 21 — WAIT HOMING COMPLETE
    //==========================================================
    21:
        // Start infeed/outfeed only after homing is complete
        IF lowerLevelStatusW1.homingComplete THEN
            lowerLevelInFeedRun  := TRUE;
            lowerLevelOutFeedRun := TRUE;
            lowerLevelStep := 40;
        END_IF

    //==========================================================
    // 40 — NORMAL OPERATION
    //==========================================================
    40:
        // Track line speed continuously
        lowerLevelInFeedDriveRef  := lineSpeedMPM;
        lowerLevelOutFeedDriveRef := lineSpeedMPM;

        // Enable cut only when commanded and paper present
        lowerLevelCut := (lowerLevelCutCmd AND lowerLevelPaperSensor);

END_CASE

//==============================================================
// 5) GLOBAL INTERLOCK — IMMEDIATE STOP
//==============================================================
// Immediate stop on any of these conditions:
// - Safety chain not OK
// - Any drive not OK
// - Power OFF command rising edge
IF (NOT safetyFeedback) OR (NOT lowerLevelAllDrivesOK) OR lowerLevelRtPowerOff.Q THEN

    lowerLevelStep := 0;

    lowerLevelEnable      := FALSE;
    lowerLevelSlave1Run   := FALSE;
    lowerLevelSlave2Run   := FALSE;
    lowerLevelInFeedRun   := FALSE;
    lowerLevelOutFeedRun  := FALSE;

    lowerLevelJogFw       := FALSE;
    lowerLevelJogRev      := FALSE;
    lowerLevelHome        := FALSE;
    lowerLevelCut         := FALSE;

    lowerLevelInFeedDriveRef  := 0.0;
    lowerLevelOutFeedDriveRef := 0.0;

    // Reset internal timers for a clean restart
    lowerLevelTimerWait(IN := FALSE);
    lowerLevelTimerPulse(IN := FALSE);
    lowerLevelTimerClear(IN := FALSE);
    lowerLevelTimerReset(IN := FALSE);
END_IF
END_METHOD

END_FUNCTION_BLOCK

// ---- Library/Machine/Slitter/FunctionBlocks/FB_PaperDirectionControl_.TcPOU
FUNCTION_BLOCK FB_PaperDirectionControl_
VAR_INPUT
	
	executeCmd	: BOOL;
	allUPCmd : BOOL;
	allDownCmd : BOOL;
	invertDirection	: BOOL;
	numberOfFlaps				: INT := 27;
	flapsManualCmdArr			: ARRAY [1..27] OF hmiCommandsFlaps_TypeStruct;	
	currentOrder				: Order_TypeStruct;
	machineConfig				: slitterConfig_TypeStruct; // Slitter configuration parameters / Parâmetros do slitter

END_VAR
VAR_OUTPUT
	
	flapSolenoidArr			: ARRAY [1..27] OF BOOL;	

END_VAR


VAR
	invertDirectionOld	: BOOL;
	executeCmdOld: BOOL;
	i: INT;
END_VAR

// Trigger logic on rising edge of execute command
IF executeCmd AND NOT executeCmdOld THEN

    FOR i := 1 TO numberOfFlaps DO
        
        // 1. Level 1 Only (Upper)
        IF currentOrder.levelSelector = E_LevelSelector.eUpperOnly THEN
            flapSolenoidArr[i] := TRUE;

        // 2. Level 2 Only (Lower)
        ELSIF currentOrder.levelSelector = E_LevelSelector.eLowerOnly THEN
            flapSolenoidArr[i] := FALSE;

        // 3. Both Levels (Decision based on Order 1 Width vs Flap physical position)
        ELSIF currentOrder.levelSelector = E_LevelSelector.eBoth THEN
            
            // If flap is within the width of Order 1, it follows Order 1 direction
            IF machineConfig.arrFlapPosition[i] <= (currentOrder.generatedOrder.order1Width + currentOrder.generatedOrder.firstKnifePosition) THEN
                flapSolenoidArr[i] :=  FALSE;
            ELSE
                // Otherwise it follows Order 2 direction
                flapSolenoidArr[i] :=  TRUE;
            END_IF;

        END_IF;
    END_FOR;

END_IF;
// Update edge detection memory
executeCmdOld := executeCmd;

// Global Overrides (Master Up / Master Down)
// These run regardless of the executeCmd rising edge if triggered
IF allUPCmd THEN
    FOR i := 1 TO 27 DO flapSolenoidArr[i] := TRUE; END_FOR;
ELSIF allDownCmd THEN
    FOR i := 1 TO 27 DO flapSolenoidArr[i] := FALSE; END_FOR;
	
END_IF;

// Manual HMI Control Override (If enabled in the HMI command structure)
FOR i := 1 TO 27 DO
    IF flapsManualCmdArr[i].upCmd THEN
        flapSolenoidArr[i] := TRUE;
    END_IF;
	
    IF flapsManualCmdArr[i].downCmd THEN
        flapSolenoidArr[i] := FALSE;
    END_IF;	
	
END_FOR;

//Invert flap direction
IF invertDirection AND NOT invertDirectionOld THEN
	
	// Loop through all flaps and flip their current solenoid state
	FOR i := 1 TO numberOfFlaps DO
		flapSolenoidArr[i] := NOT flapSolenoidArr[i];
	END_FOR;

END_IF
invertDirectionOld := invertDirection;

END_FUNCTION_BLOCK

// ---- Library/Machine/Slitter/FunctionBlocks/FB_SpeedMeter.TcPOU
FUNCTION_BLOCK FB_SpeedMeter
VAR_INPUT

	mesuringWheelPulseSensor		: BOOL;
	measuringWheelDiameter		: REAL	:= 159.0;
	cycleTimeSeconds			: TIME	:= T#1S;

END_VAR
VAR_OUTPUT

	mesuringWheelSpeedRPM		: REAL;
	measuringWheelSpeedMPM		: REAL;

END_VAR
VAR

	measuringWheelPulseCounter	: DINT;
	measuringWheelPulseCounterOld	: DINT;
	measuringWheelPulseDif		: DINT;
	cycleCounter				: DINT;

	mesuringWheelPulseSensorOld	: BOOL;
	timerPulse					: BOOL;
	timerPulseOld				: BOOL;
	instTimerTON				: TON;

	cycleTimeSecondsInt: INT;
END_VAR



VAR CONSTANT

	PI						: REAL	:= 3.14159265359;

END_VAR



IF mesuringWheelPulseSensor AND NOT mesuringWheelPulseSensorOld THEN

	measuringWheelPulseCounter := measuringWheelPulseCounter + 1;

END_IF

mesuringWheelPulseSensorOld := mesuringWheelPulseSensor;




IF instTimerTON.Q THEN

	timerPulse := FALSE;
	instTimerTON.IN	:= FALSE;

END_IF

IF NOT instTimerTON.IN AND NOT instTimerTON.Q THEN

	timerPulse := TRUE;
	instTimerTON.PT := cycleTimeSeconds;
	instTimerTON.IN	:= TRUE;

END_IF


IF timerPulse AND NOT timerPulseOld THEN

	measuringWheelPulseDif := measuringWheelPulseCounter - measuringWheelPulseCounterOld;
	cycleCounter := cycleCounter + 1;
	measuringWheelPulseCounterOld := measuringWheelPulseCounter;

END_IF

timerPulseOld := timerPulse;

cycleTimeSecondsInt := TIME_TO_INT(cycleTimeSeconds / 1000);

mesuringWheelSpeedRPM := (60 / cycleTimeSecondsInt) * measuringWheelPulseDif;

measuringWheelSpeedMPM :=  (mesuringWheelSpeedRPM * ( measuringWheelDiameter * PI)*0.001);


instTimerTON();

END_FUNCTION_BLOCK

// ---- Library/Machine/Stacker/Cpx/FB_ComplexSheetStackerControl_1.TcPOU
FUNCTION_BLOCK FB_ComplexSheetStackerControl_1
VAR_INPUT

    //==============================================================
    // Group command inputs
    //==============================================================
    startCmd                            : BOOL;
    stopCmd                             : BOOL;
    resetCmd                            : BOOL;


    //==============================================================
    // Speed reference inputs
    //==============================================================
    lineSpeedMPM                        : REAL;

    // EN: Current sheet length [mm].
    // PT: Comprimento atual da chapa [mm].
    sheetLengthMm                       : REAL;


    //==============================================================
    // Package command input
    //==============================================================
    // EN: Rising edge starts package separation cycle.
    // PT: Borda de subida inicia o ciclo de separação do pacote.
    packageCompleteCmd                  : BOOL;
	sheetConveyorsSpeedUpCmd : BOOL;

    //==============================================================
    // Machine configuration
    //==============================================================
    machineConfig                       : ComplexStackerConfig_TypeStruct;


    //==============================================================
    // Safety input
    //==============================================================
    safetyCircuitOk                     : BOOL;


    //==============================================================
    // Synchronized conveyor drive status inputs
    //==============================================================
    sheetConveyor1DriveOk               : BOOL;
    sheetConveyor2DriveOk               : BOOL;
    sheetConveyor3DriveOk               : BOOL;
    sheetConveyor4DriveOk               : BOOL;
    elevatorDriveOk              : BOOL;


    //==============================================================
    // Auxiliary drive status inputs
    //==============================================================
    backstopDriveOk                     : BOOL;

	//==============================================================
	// Sheet stack discharge conveyor drive status input
	//==============================================================
    sheetStackDischargeConveyorDriveOk                 : BOOL;

	//==============================================================
	// EN: Stack buffer conveyor drive status inputs
	// PT: Entradas de estado dos acionamentos das esteiras buffer
	//==============================================================
	stackBufferConveyor1DriveOk            : BOOL;
	stackBufferConveyor2DriveOk            : BOOL;
	stackBufferConveyor3DriveOk            : BOOL;

	//==============================================================
	// EN: Stack detection sensors
	// PT: Sensores de detecção das pilhas
	//==============================================================
	stackBufferConveyor1StackPresentSensor : BOOL;
	stackBufferConveyor2StackPresentSensor : BOOL;
	stackBufferConveyor3StackPresentSensor : BOOL;
	elevatorStackPresentSensor             : BOOL;
	elevatorStackExitClearSensor           : BOOL;
	backstopMaterialInterlockSensor         : BOOL;
	backstopStackLevelSensor                : BOOL;

	
    //==============================================================
    // Position / measurement inputs
    //==============================================================
    stackHeightMm                       : REAL;
    backstopPositionMm                  : REAL;
    elevatorPositionMm           : REAL;


	//==============================================================
	// Elevator command inputs
	//==============================================================
	// EN: Starts elevator homing cycle.
	// PT: Inicia o ciclo de homing do elevador.
	elevatorHomeCmd              : BOOL;
	
	// EN: Enables elevator automatic mode. Auto-home is requested on
	//     startCmd and automatic leveling uses the stack level sensor.
	// PT: Habilita o modo automático do elevador. O auto-home é solicitado
	//     no startCmd e o nivelamento automático usa o sensor de nível da pilha.
	elevatorAutoCmd              : BOOL;
	
	// EN: Jog-up command in manual mode or during automatic leveling.
	// PT: Comando de jog para subir no manual ou durante o nivelamento automático.
	elevatorUpCmd                : BOOL;
	
	// EN: Jog-down command in manual mode or during automatic leveling.
	// PT: Comando de jog para descer no manual ou durante o nivelamento automático.
	elevatorDownCmd              : BOOL;


    //==============================================================
    // Elevator limit inputs
    //==============================================================
    elevatorUpperSafetyLimit     : BOOL;
    elevatorLowerSafetyLimit     : BOOL;

    elevatorUpperLimit           : BOOL;
    elevatorLowerLimit           : BOOL;


    //==============================================================
    // Backstop command inputs
    //==============================================================
    // EN: Starts the backstop homing cycle.
    // PT: Inicia o ciclo de homing do backstop.
    backstopHomeCmd                     : BOOL;
	
    // EN: Starts the backstop homing cycle.
    // PT: Inicia o ciclo de homing do backstop.
    backstopExecutePositioningCmd			 : BOOL;
    // EN: Enables automatic positioning according to sheet length.
    // PT: Habilita posicionamento automático conforme comprimento da chapa.
    backstopAutoCmd                     : BOOL;

    // EN: Manual open command.
    // PT: Comando manual para abrir.
    backstopOpenCmd                     : BOOL;

    // EN: Manual close command.
    // PT: Comando manual para fechar.
    backstopCloseCmd                    : BOOL;


    //==============================================================
    // Backstop limit inputs
    //==============================================================
    backstopSafeMaxLimit                    : BOOL;	
    backstopMaxLimit                 	   	: BOOL;
    backstopMinLimit                   		: BOOL;
    backstopSafeMinLimit                    : BOOL;


    //==============================================================
    // Sheet handling command inputs
    //==============================================================
	sheetStackDischargeConveyorManualRunCmd : BOOL;
    noCrushRollersDownCmd                 	: BOOL;

	// EN: Runs all three stack buffer conveyors.
	// PT: Aciona as três esteiras buffer de pilhas.
	stackBufferConveyorsRunCmd               : BOOL;

END_VAR


VAR_OUTPUT

	hmiAlarms : hmiAlarmsComplexStacker_TypeStruct;
	hmiStatus : hmiStatusComplexStacker_TypeStruct;
	stackerRunning : BOOL;
	alarmActive	: BOOL;
	stopMachinePulse : BOOL;
	reset 	: BOOL;
    //==============================================================
    // Synchronized conveyor drive outputs
    //==============================================================
    sheetConveyor1Run                   : BOOL;
    sheetConveyor2Run                   : BOOL;
    sheetConveyor3Run                   : BOOL;
    sheetConveyor4Run                   : BOOL;
	
	//==============================================================
	// Elevator drive outputs
	//==============================================================
	// EN: Elevator up run command.
	// PT: Comando para subir o elevador.
	elevatorRunUp                : BOOL;
	
	// EN: Elevator down run command.
	// PT: Comando para descer o elevador.
	elevatorRunDown              : BOOL;
	
	//==============================================================
	// Elevator magnetic brake output
	//==============================================================
	// EN: Magnetic brake release output. TRUE = brake released.
	// PT: Saída de liberação do freio magnético. TRUE = freio liberado.
	elevatorBrakeRelease         : BOOL;	

	// EN: Enables the elevator servo together with the stacker control.
	//     The servo remains enabled while stopped with zero speed reference.
	// PT: Habilita o servo do elevador junto com o controle do stacker.
	//     O servo permanece habilitado quando parado com referência zero.
	elevatorDriveEnable          : BOOL;

    //==============================================================
    // Backstop drive outputs
    //==============================================================
    // EN: Backstop forward run command. Positive/opening direction.
    // PT: Comando frente do backstop. Direção positiva/abrir.
    backstopRunFw                       : BOOL;

    // EN: Backstop reverse run command. Negative/closing direction.
    // PT: Comando reverso do backstop. Direção negativa/fechar.
    backstopRunRev                      : BOOL;

    // EN: Enables the backstop servo together with the stacker control.
    // PT: Habilita o servo do backstop junto com o controle do stacker.
    backstopDriveEnable                 : BOOL;

	//==============================================================
	// Sheet stack discharge conveyor outputs
	//==============================================================
	// EN: Sheet stack discharge conveyor run command.
	// PT: Comando de giro da esteira de descarga da pilha.
	sheetStackDischargeConveyorRun          : BOOL;

	//==============================================================
	// EN: Stack buffer conveyor run outputs
	// PT: Saídas de acionamento das esteiras buffer de pilhas
	//==============================================================
	stackBufferConveyor1Run                 : BOOL;
	stackBufferConveyor2Run                 : BOOL;
	stackBufferConveyor3Run                 : BOOL;




    //==============================================================
    // Synchronized conveyor speed reference outputs
    //==============================================================
    sheetConveyor1SpeedRefMPM           : REAL;
    sheetConveyor2SpeedRefMPM           : REAL;
    sheetConveyor3SpeedRefMPM           : REAL;
    sheetConveyor4SpeedRefMPM           : REAL;

    // EN: Signed elevator speed reference [mm/s]. Positive moves up
    //     and negative moves down.
    // PT: Referência de velocidade com sinal do elevador [mm/s].
    //     Positivo sobe e negativo desce.
    elevatorSpeedRefMmps                 : REAL;
	// EN: Sheet stack discharge conveyor speed reference [m/min].
	// PT: Referência de velocidade da esteira de descarga da pilha [m/min].
	sheetStackDischargeConveyorSpeedRefMPM  : REAL;

	// EN: Stack buffer conveyor speed references [m/min].
	// PT: Referências de velocidade das esteiras buffer [m/min].
	stackBufferConveyor1SpeedRefMPM         : REAL;
	stackBufferConveyor2SpeedRefMPM         : REAL;
	stackBufferConveyor3SpeedRefMPM         : REAL;

	// EN: TRUE while all three stack buffer positions are occupied.
	// PT: TRUE enquanto as três posições buffer estiverem ocupadas.
	stackBufferFull                         : BOOL;

	// EN: Requests the parent controller to reduce the machine speed.
	// PT: Solicita ao controlador pai a redução da velocidade da máquina.
	lineSpeedReductionRequest               : BOOL;

    //==============================================================
    // Backstop speed reference output
    //==============================================================
    // EN: Signed backstop speed reference [mm/s]. Positive opens and negative closes.
    // PT: Referência de velocidade com sinal do backstop [mm/s]. Positivo abre e negativo fecha.
    backstopSpeedRefMmps                : REAL;
	
	
	
    backstopPlateUpSolenoid                : BOOL;


    //==============================================================
    // Backstop encoder set outputs
    //==============================================================
    // EN: Pulse output to set/reset backstop encoder position.
    // PT: Pulso de saída para setar/resetar a posição do encoder do backstop.
    backstopSetEncoderPosition          : BOOL;

    // EN: Position value to set in the encoder block [mm].
    // PT: Valor de posição a ser gravado no bloco do encoder [mm].
    backstopSetEncoderPositionMm        : REAL;


    //==============================================================
    // Pneumatic valve outputs
    //==============================================================
    brakeValve                          : BOOL;

    sheetBrush1Valve                    : BOOL;
    sheetBrush2Valve                    : BOOL;
    sheetBrush3Valve                    : BOOL;

    brakeBrushValve                     : BOOL;
    backstopUpValve                     : BOOL;
    noCrushRollersUpDownValve               : BOOL;


    //==============================================================
    // General status outputs
    //==============================================================
    deviceState                         : STRING(30);

    faultActive                         : BOOL;
    synchronizedConveyorsRunning        : BOOL;


    //==============================================================
    // Sheet stack separation status outputs
    //==============================================================
    sheetStackSeparationState           : STRING(30);
    sheetStackSeparationStateCode       : INT;

    sheetStackSeparationReady           : BOOL;
    sheetStackSeparationActive          : BOOL;

    // EN: One-scan pulse when sheet stack separation starts.
    // PT: Pulso de um ciclo quando inicia a separação da pilha de chapas.
    sheetStackSeparationStarted         : BOOL;

    // EN: One-scan pulse when sheet stack separation finishes.
    // PT: Pulso de um ciclo quando finaliza a separação da pilha de chapas.
    sheetStackSeparationFinished        : BOOL;

    // EN: Brake active during sheet stack separation.
    // PT: Freio ativo durante a separação da pilha de chapas.
    sheetStackBrakeActive               : BOOL;


    //==============================================================
    // Sheet conveyor 2 separation status outputs
    //==============================================================
    sheetConveyor2SeparationActive      : BOOL;

    // EN: One-scan pulse when conveyor 2 separation tracking starts.
    // PT: Pulso de um ciclo quando inicia o rastreamento de separação da esteira 2.
    sheetConveyor2SeparationStarted     : BOOL;

    // EN: One-scan pulse when conveyor 2 separation tracking finishes.
    // PT: Pulso de um ciclo quando finaliza o rastreamento de separação da esteira 2.
    sheetConveyor2SeparationFinished    : BOOL;

    sheetConveyor2HighSpeedActive       : BOOL;

    // EN: Current conveyor 2 separation tracking distance [m].
    // PT: Distância atual rastreada na separação da esteira 2 [m].
    sheetConveyor2TrackingDistanceM     : REAL;

    // EN: Conveyor 2 separation target distance [m].
    // PT: Distância alvo de separação da esteira 2 [m].
    sheetConveyor2TargetDistanceM       : REAL;


    //==============================================================
    // Sheet conveyor 3 separation status outputs
    //==============================================================
    sheetConveyor3SeparationActive      : BOOL;

    // EN: One-scan pulse when conveyor 3 separation tracking starts.
    // PT: Pulso de um ciclo quando inicia o rastreamento de separação da esteira 3.
    sheetConveyor3SeparationStarted     : BOOL;

    // EN: One-scan pulse when conveyor 3 separation tracking finishes.
    // PT: Pulso de um ciclo quando finaliza o rastreamento de separação da esteira 3.
    sheetConveyor3SeparationFinished    : BOOL;

    sheetConveyor3HighSpeedActive       : BOOL;

    // EN: Current conveyor 3 separation tracking distance [m].
    // PT: Distância atual rastreada na separação da esteira 3 [m].
    sheetConveyor3TrackingDistanceM     : REAL;

    // EN: Conveyor 3 separation target distance [m].
    // PT: Distância alvo de separação da esteira 3 [m].
    sheetConveyor3TargetDistanceM       : REAL;

    //==============================================================
    // Sheet conveyor 4 separation status outputs
    //==============================================================
    sheetConveyor4SeparationActive      : BOOL;
    sheetConveyor4SeparationStarted     : BOOL;
    sheetConveyor4SeparationFinished    : BOOL;
    sheetConveyor4HighSpeedActive       : BOOL;
    sheetConveyor4TrackingDistanceM     : REAL;
    sheetConveyor4TargetDistanceM       : REAL;

	//==============================================================
	// Elevator encoder set outputs
	//==============================================================
	// EN: Pulse output to set/reset elevator encoder position.
	// PT: Pulso de saída para setar/resetar a posição do encoder do elevador.
	elevatorSetEncoderPosition   : BOOL;
	
	// EN: Position value to set in the elevator encoder block [mm].
	// PT: Valor de posição a ser gravado no bloco do encoder do elevador [mm].
	elevatorSetEncoderPositionMm : REAL;
	
	
	//==============================================================
	// Elevator status outputs
	//==============================================================
	elevatorState                : STRING(30);
	
	elevatorHomed                : BOOL;
	elevatorInPosition           : BOOL;

	// EN: TRUE when the homed elevator is at or below the configured
	//     minimum position considering the position tolerance.
	// PT: TRUE quando o elevador referenciado está na posição mínima
	//     configurada ou abaixo dela, considerando a tolerância.
	elevatorAtMinPosition        : BOOL;

	// EN: TRUE when the homed elevator is at or above the configured
	//     maximum position considering the position tolerance.
	// PT: TRUE quando o elevador referenciado está na posição máxima
	//     configurada ou acima dela, considerando a tolerância.
	elevatorAtMaxPosition        : BOOL;

	// EN: TRUE while manual jog speed is reduced near the endpoint
	//     toward which the elevator is moving.
	// PT: TRUE enquanto a velocidade do jog manual estiver reduzida próximo
	//     da extremidade para a qual o elevador está se movimentando.
	elevatorManualLowSpeedZoneActive : BOOL;

	elevatorFault                : BOOL;
	elevatorFaultCode            : INT;
	
	// EN: Current calculated elevator target position [mm].
	// PT: Posição alvo calculada atual do elevador [mm].
	elevatorTargetPositionMm     : REAL;
	
	// EN: Current elevator position error [mm].
	// PT: Erro atual de posição do elevador [mm].
	elevatorPositionErrorMm      : REAL;

    //==============================================================
    // Backstop status outputs
    //==============================================================
    backstopState                       : STRING(30);

    backstopHomed                       : BOOL;
    backstopInPosition                  : BOOL;
    backstopFault                       : BOOL;
    backstopFaultCode                   : INT;

    // EN: Current calculated target position [mm].
    // PT: Posição alvo calculada atualmente [mm].
    backstopTargetPositionMm            : REAL;

    // EN: Current position error [mm].
    // PT: Erro atual de posição [mm].
    backstopPositionErrorMm             : REAL;
	
	//==============================================================
	// Sheet stack discharge conveyor control state
	//==============================================================
	sheetStackDischargeConveyorState               : STRING(30);
	sheetStackDischargeConveyorFault               : BOOL;
	sheetStackDischargeConveyorFaultCode           : INT;
	
	//==============================================================
	// Sheet stack discharge sequence status outputs
	//==============================================================
	sheetStackDischargeState                : STRING(30);
	sheetStackDischargeStateCode            : INT;
	
	sheetStackDischargePending              : BOOL;
	sheetStackDischargeActive               : BOOL;
	sheetStackDischargeStarted              : BOOL;
	sheetStackDischargeFinished             : BOOL;
	
	sheetStackDischargeFault                : BOOL;
	sheetStackDischargeFaultCode            : INT;
	
	//==============================================================
	// Sheet stack discharge last cycle diagnostic outputs
	//==============================================================
	sheetStackDischargeLastCycleOk          : BOOL;
	sheetStackDischargeLastResultCode       : INT;
	sheetStackDischargeLastFaultStepCode    : INT;
	sheetStackDischargeLastFaultCode        : INT;	

END_VAR

VAR
	
	//==============================================================
	// Stop machine pulse control
	//==============================================================
	stopMachineFaultCondition     : BOOL;
	stopMachineFaultConditionOld  : BOOL;
	rStopMachineFaultCondition    : BOOL;
	
	tpStopMachinePulse            : TP;
	
	//==============================================================
	// Backstop manual intervention memory
	//==============================================================
	backstopManualInterventionActive     : BOOL;
	backstopManualInterventionPositionMm : REAL;
	
	//==============================================================
	// Sheet stack discharge backstop latched targets
	//==============================================================
	backstopProgrammedDischargeTargetMm : REAL;
	backstopDischargeOpenBasePositionMm : REAL;
	backstopDischargeOpenTargetMm       : REAL;
	
	//==============================================================
	// Backstop automatic positioning command control
	//==============================================================
	backstopExecutePositioningCmdOld    : BOOL;
	rBackstopExecutePositioning         : BOOL;
	
	backstopTargetOverrideOld           : BOOL;
	backstopTargetOverrideFallingEdge   : BOOL;
	
	backstopPositioningRequestActive    : BOOL;
	backstopLatchedTargetPositionMm     : REAL;
	backstopProgrammedTargetPositionMm  : REAL;
	
	//==============================================================
	// Backstop manual intervention memory
	//==============================================================
	// EN: Used by automatic discharge sequence to avoid closing onto material
	//     after operator manual intervention.

	//==============================================================
	// Backstop encoder set pulse
	//==============================================================
	backstopSetEncoderPositionTrigger  : BOOL;
	tpBackstopSetEncoderPosition       : TP;

	//==============================================================
	// Sheet stack discharge backstop latched targets
	//==============================================================

    //==============================================================
    // Group state machine
    //==============================================================
    syncConveyorsState                  : INT;


    //==============================================================
    // Package separation state machine
    //==============================================================
    packageSeparationState              : INT;


    //==============================================================
    // Backstop state machine
    //==============================================================
    backstopControlState                : INT;


    //==============================================================
    // Edge detection
    //==============================================================
    startCmdOld                         : BOOL;
    stopCmdOld                          : BOOL;
    packageCompleteCmdOld               : BOOL;

    backstopHomeCmdOld                  : BOOL;


    //==============================================================
    // Internal conditions
    //==============================================================
    allSynchronizedDrivesOk             : BOOL;
    anyFault                            : BOOL;
    speedControlEnabled                 : BOOL;
    rampReset                           : BOOL;


    //==============================================================
    // Sheet length conversion
    //==============================================================
    // EN: Internal sheet length converted from mm to m.
    // PT: Comprimento interno da chapa convertido de mm para m.
    sheetLengthM                        : REAL;


    //==============================================================
    // Normal speed calculation
    //==============================================================
    normalStackerSpeedMPM               : REAL;

    sheetConveyor1NormalSpeedMPM        : REAL;
    sheetConveyor2NormalSpeedMPM        : REAL;
    sheetConveyor3NormalSpeedMPM        : REAL;
    sheetConveyor4NormalSpeedMPM        : REAL;
    elevatorNormalSpeedMPM       : REAL;


    //==============================================================
    // Package gap speed calculation
    //==============================================================
    sheetConveyor2GapSpeedMPM           : REAL;
    sheetConveyor3GapSpeedMPM           : REAL;
    sheetConveyor4GapSpeedMPM           : REAL;


    //==============================================================
    // Speed targets
    //==============================================================
    sheetConveyor1TargetSpeedMPM        : REAL;
    sheetConveyor2TargetSpeedMPM        : REAL;
    sheetConveyor3TargetSpeedMPM        : REAL;
    sheetConveyor4TargetSpeedMPM        : REAL;
    elevatorTargetSpeedMPM       : REAL;


    //==============================================================
    // Package gap distance calculation
    //==============================================================
    packageGapDistanceTargetM           : REAL;

    sheetConveyor2OpeningSpeedMPM       : REAL;
    sheetConveyor3OpeningSpeedMPM       : REAL;
    sheetConveyor4OpeningSpeedMPM       : REAL;

    sheetConveyor2OpeningDistanceM      : REAL;
    sheetConveyor3OpeningDistanceM      : REAL;
    sheetConveyor4OpeningDistanceM      : REAL;


	//==============================================================
	// Elevator state machine
	//==============================================================
	elevatorControlState         : INT;
	
	
	//==============================================================
	// Elevator edge detection
	//==============================================================
	elevatorHomeCmdOld           : BOOL;
	rElevatorHome                : BOOL;
	
	
	//==============================================================
	// Elevator encoder set pulse
	//==============================================================
	elevatorSetEncoderPositionTrigger   : BOOL;
	tpElevatorSetEncoderPosition        : TP;
	
	
	//==============================================================
	// Elevator control calculation
	//==============================================================
	elevatorAutoTargetPositionMm        : REAL;
	elevatorRawSpeedRefMmps             : REAL;
	
	// EN: Internal signed speed command. Positive = up, negative = down.
	// PT: Comando interno de velocidade com sinal. Positivo = subir, negativo = descer.
	elevatorSignedSpeedRefMmps          : REAL;
	
	elevatorAbsPositionErrorMm          : REAL;
	
	
	//==============================================================
	// Elevator movement permissions
	//==============================================================
	elevatorUpAllowed                   : BOOL;
	elevatorDownAllowed                 : BOOL;
	
	elevatorMoveRequest                 : BOOL;
	elevatorBrakeReleaseRequest         : BOOL;
	
	
	//==============================================================
	// Elevator homing
	//==============================================================
	elevatorHomeLimitReached            : BOOL;
	elevatorHomeDownAllowed             : BOOL;
	elevatorHomeReleaseAllowed          : BOOL;
	elevatorManualCommandArmed          : BOOL;
	elevatorManualCommandRequest        : BOOL;
	elevatorReadyForAutomaticCycle      : BOOL;
	
	
	//==============================================================
	// Elevator timers
	//==============================================================
	tonElevatorHomingTimeout            : TON;
	tonElevatorHomeSettleDelay          : TON;
	tonElevatorLevelingSpeed2Delay      : TON;
	
	// EN: Delay after brake release before motor movement.
	// PT: Atraso após liberar o freio antes de movimentar o motor.
	tonElevatorBrakeReleaseDelay        : TON;
	
	// EN: Keeps brake released for a short time after movement stops.
	// PT: Mantém o freio liberado por um tempo após parar o movimento.
	tonElevatorBrakeHoldDelay           : TON;
	
	
	//==============================================================
	// Elevator speed ramp instance
	//==============================================================
	// EN: Ramp used for elevator vertical speed [mm/s].
	// PT: Rampa usada para velocidade vertical do elevador [mm/s].
	instRampElevator                    : FB_Gen_SRamp;
	

    //==============================================================
    // Backstop control calculation
    //==============================================================
    backstopAutoTargetPositionMm        : REAL;
    backstopRawSpeedRefMmps             : REAL;
    backstopAbsPositionErrorMm          : REAL;

    backstopHomeLimitReached            : BOOL;
    backstopOpenAllowed                 : BOOL;
    backstopCloseAllowed                : BOOL;

    rBackstopHome                       : BOOL;


	//==============================================================
	// Backstop homing edge detection
	//==============================================================
	backstopHomeLimitOld                 : BOOL;
	backstopHomeLimitFallingEdge         : BOOL;
	backstopHomeMoveAllowed              : BOOL;
	
	
	
	//==============================================================
	// Backstop timers
	//==============================================================
	tonBackstopHomeSettleDelay           : TON;



    //==============================================================
    // Backstop timers
    //==============================================================
    tonBackstopHomingTimeout            : TON;


    //==============================================================
    // Speed ramp instances
    //==============================================================
    instRampSheetConveyor1              : FB_Gen_SRamp;
    instRampSheetConveyor2              : FB_Gen_SRamp;
    instRampSheetConveyor3              : FB_Gen_SRamp;
    instRampSheetConveyor4              : FB_Gen_SRamp;


    //==============================================================
    // PLC scan time measurement
    //==============================================================
    instCycleTime                       : CYCLE_TIME;
    scanTimeS                           : REAL;
    scanTimeMs                          : REAL;

	backstopSignedSpeedRefMmps: REAL;
	
	//==============================================================
	// Sheet stack discharge state machine
	//==============================================================
	sheetStackDischargeControlState         : INT;
	
	
	//==============================================================
	// Sheet stack discharge edge detection
	//==============================================================
	packageCompleteCmdOldDischarge          : BOOL;
	rPackageCompleteDischarge               : BOOL;
	
	
	//==============================================================
	// Sheet stack discharge timers
	//==============================================================
	tonSheetStackDischarge                  : TON;
	tonSheetStackDischargePlatformClearTimeout : TON;
	elevatorPlatformClearDetected           : BOOL;
	elevatorStackPresentAtDischargeStart    : BOOL;
	
	
	//==============================================================
	// Sheet stack discharge internal conditions
	//==============================================================
	sheetStackDischargeFaultCondition       : BOOL;
	
	
	//==============================================================
	// Backstop target override
	//==============================================================
	backstopTargetOverrideActive            : BOOL;
	backstopTargetOverridePositionMm        : REAL;
	
	
	//==============================================================
	// Elevator target override
	//==============================================================
	elevatorTargetOverrideActive     : BOOL;
	elevatorTargetOverridePositionMm : REAL;	
	
	
	sheetStackDischargeConveyorRunRequest: BOOL;
	instTONBackstopDownDelay: TON;
	
	//==============================================================
	// Sheet stack discharge step timeout
	//==============================================================
	tonSheetStackDischargeStepTimeout       : TON;
	
	sheetStackDischargeCycleHasManualSkip   : BOOL;
	sheetStackDischargeCycleHasTimeout      : BOOL;	
	
	
	//==============================================================
	// Elevator homing edge detection
	//==============================================================
	elevatorHomeLimitOld                 : BOOL;
	elevatorHomeLimitFallingEdge         : BOOL;	

	//==============================================================
	// System master run control
	//==============================================================
	systemRunEnable : BOOL;
	
	rStartCmd : BOOL;
	rStopCmd  : BOOL;
	
	//==============================================================
	// Automatic homing requests generated by master start
	//==============================================================
	backstopAutoHomeRequest        : BOOL;
	elevatorAutoHomeRequest : BOOL;
	
	//==============================================================
	// Elevator home request command control
	//==============================================================
	elevatorHomeRequestCombined    : BOOL;
	elevatorHomeRequestCombinedOld : BOOL;
	backstopHomeRunning: BOOL;
	//==============================================================
	// Backstop home request command control
	//==============================================================
	backstopHomeRequestCombined    : BOOL;
	backstopHomeRequestCombinedOld : BOOL;

	//==============================================================
	// EN: Stack buffer conveyor control
	// PT: Controle das esteiras buffer de pilhas
	//==============================================================
	stackBufferControlState                 : INT;
	stackBufferTargetConveyor               : INT;
	elevatorStackExitClearSensorOld         : BOOL;
	rElevatorStackExitClear                 : BOOL;
	tonStackBufferStopDelay                 : TON;
	tonStackBufferTransferTimeout           : TON;
	tonStackBufferFullSpeedReduction        : TON;
	
END_VAR

_SystemControl();

_SheetConveyorGroupControl();
_ConveyorSpeedControl();

_SheetStackDischargeControl();

_BackstopControl();
_ElevatorControl();
_SheetStackDischargeConveyorControl();
_StackBufferConveyorsControl();
_MachineAuxilary();
_HmiStatus();
_AlarmControl();

//==============================================================
// COMPLEX STACKER — ALARM CONTROL
// EN: Maps internal faults and status conditions to HMI alarm structure.
//==============================================================
METHOD _AlarmControl

VAR
	hmiAlarmsNotActive: hmiAlarmsComplexStacker_TypeStruct;
END_VAR
//==============================================================
// HMI alarms reset / latch logic
//==============================================================

IF resetCmd THEN

    // Reset geral dos alarmes
    hmiAlarms := hmiAlarmsNotActive;

ELSE

    //==============================================================
    // 1) General / system alarms
    //==============================================================
    hmiAlarms.safetyCircuitNotOk :=
        hmiAlarms.safetyCircuitNotOk OR
        NOT safetyCircuitOk;

    hmiAlarms.systemFaultActive :=
        hmiAlarms.systemFaultActive OR
        faultActive OR
        backstopFault OR
        elevatorFault OR
        sheetStackDischargeFault OR
        sheetStackDischargeConveyorFault OR
        NOT stackBufferConveyor1DriveOk OR
        NOT stackBufferConveyor2DriveOk OR
        NOT stackBufferConveyor3DriveOk;

    hmiAlarms.systemNotEnabled :=
        hmiAlarms.systemNotEnabled OR
        NOT systemRunEnable;


    //==============================================================
    // 2) Sheet conveyor group alarms
    //==============================================================
    hmiAlarms.sheetConveyor1DriveNotOk :=
        hmiAlarms.sheetConveyor1DriveNotOk OR
        NOT sheetConveyor1DriveOk;

    hmiAlarms.sheetConveyor2DriveNotOk :=
        hmiAlarms.sheetConveyor2DriveNotOk OR
        NOT sheetConveyor2DriveOk;

    hmiAlarms.sheetConveyor3DriveNotOk :=
        hmiAlarms.sheetConveyor3DriveNotOk OR
        NOT sheetConveyor3DriveOk;

    hmiAlarms.sheetConveyor4DriveNotOk :=
        hmiAlarms.sheetConveyor4DriveNotOk OR
        NOT sheetConveyor4DriveOk;

    hmiAlarms.sheetConveyorGroupFault :=
        hmiAlarms.sheetConveyorGroupFault OR
        NOT safetyCircuitOk OR
        NOT sheetConveyor1DriveOk OR
        NOT sheetConveyor2DriveOk OR
        NOT sheetConveyor3DriveOk OR
        NOT sheetConveyor4DriveOk;


    //==============================================================
    // 2.1) Stack buffer conveyor alarms
    // EN: Buffer drive faults are alarmed without stopping the main
    //     synchronized conveyor group automatically.
    // PT: Falhas dos drives do buffer geram alarme sem parar automaticamente
    //     o grupo principal de esteiras sincronizadas.
    //==============================================================
    hmiAlarms.stackBufferConveyor1DriveNotOk :=
        hmiAlarms.stackBufferConveyor1DriveNotOk OR
        NOT stackBufferConveyor1DriveOk;

    hmiAlarms.stackBufferConveyor2DriveNotOk :=
        hmiAlarms.stackBufferConveyor2DriveNotOk OR
        NOT stackBufferConveyor2DriveOk;

    hmiAlarms.stackBufferConveyor3DriveNotOk :=
        hmiAlarms.stackBufferConveyor3DriveNotOk OR
        NOT stackBufferConveyor3DriveOk;

    hmiAlarms.stackBufferConveyorGroupFault :=
        hmiAlarms.stackBufferConveyorGroupFault OR
        NOT safetyCircuitOk OR
        NOT stackBufferConveyor1DriveOk OR
        NOT stackBufferConveyor2DriveOk OR
        NOT stackBufferConveyor3DriveOk;

 //   hmiAlarms.synchronizedConveyorsNotRunning :=
 //       hmiAlarms.synchronizedConveyorsNotRunning OR
 //       (
 //           systemRunEnable AND
 //           NOT synchronizedConveyorsRunning
 //       );


    //==============================================================
    // 3) Sheet stack separation alarms / indications
    //==============================================================
    // Mantido comentado conforme lógica original.
    // Se quiser ativar como latch, use o mesmo padrão:
    //
    // hmiAlarms.sheetStackSeparationNotReady :=
    //     hmiAlarms.sheetStackSeparationNotReady OR
    //     (
    //         systemRunEnable AND
    //         synchronizedConveyorsRunning AND
    //         NOT sheetStackSeparationReady
    //     );
    //
    // hmiAlarms.sheetStackSeparationActive :=
    //     hmiAlarms.sheetStackSeparationActive OR
    //     sheetStackSeparationActive;
    //
    // hmiAlarms.sheetStackBrakeActive :=
    //     hmiAlarms.sheetStackBrakeActive OR
    //     sheetStackBrakeActive;


    //==============================================================
    // 4) Sheet stack discharge sequence alarms / indications
    //==============================================================
    hmiAlarms.sheetStackDischargeFault :=
        hmiAlarms.sheetStackDischargeFault OR
        sheetStackDischargeFault;

    hmiAlarms.sheetStackDischargeLastCycleNotOk :=
        hmiAlarms.sheetStackDischargeLastCycleNotOk OR
        (
            NOT sheetStackDischargeLastCycleOk AND
            sheetStackDischargeLastResultCode <> 0
        );

    hmiAlarms.sheetStackDischargeTimeout :=
        hmiAlarms.sheetStackDischargeTimeout OR
        sheetStackDischargeLastResultCode = 3;

    hmiAlarms.sheetStackDischargeManualSkip :=
        hmiAlarms.sheetStackDischargeManualSkip OR
        sheetStackDischargeLastResultCode = 2;


    //==============================================================
    // 5) Sheet stack discharge conveyor alarms
    //==============================================================
    hmiAlarms.sheetStackDischargeConveyorDriveNotOk :=
        hmiAlarms.sheetStackDischargeConveyorDriveNotOk OR
        NOT sheetStackDischargeConveyorDriveOk;

    hmiAlarms.sheetStackDischargeConveyorFault :=
        hmiAlarms.sheetStackDischargeConveyorFault OR
        sheetStackDischargeConveyorFault;


    //==============================================================
    // 6) Backstop alarms / indications
    //==============================================================
    hmiAlarms.backstopDriveNotOk :=
        hmiAlarms.backstopDriveNotOk OR
        NOT backstopDriveOk;

    hmiAlarms.backstopFault :=
        hmiAlarms.backstopFault OR
        backstopFault;

    hmiAlarms.backstopNotHomed :=
        hmiAlarms.backstopNotHomed OR
        (
            backstopAutoCmd AND
            NOT backstopHomed
        );

    (*
    hmiAlarms.backstopNotInPosition :=
        hmiAlarms.backstopNotInPosition OR
        (
            systemRunEnable AND
            backstopAutoCmd AND
            backstopHomed AND
            NOT backstopInPosition AND
            NOT backstopTargetOverrideActive
        );
    *)

    hmiAlarms.backstopSafeMaxLimitActive :=
        hmiAlarms.backstopSafeMaxLimitActive OR
        backstopSafeMaxLimit;

    hmiAlarms.backstopSafeMinLimitActive :=
        hmiAlarms.backstopSafeMinLimitActive OR
        backstopSafeMinLimit;

    (*
    hmiAlarms.backstopMaxLimitActive :=
        hmiAlarms.backstopMaxLimitActive OR
        backstopMaxLimit;

    hmiAlarms.backstopMinLimitActive :=
        hmiAlarms.backstopMinLimitActive OR
        backstopMinLimit;

    hmiAlarms.backstopManualInterventionActive :=
        hmiAlarms.backstopManualInterventionActive OR
        backstopManualInterventionActive;
    *)


    //==============================================================
    // 7) Elevator alarms / indications
    //==============================================================
    hmiAlarms.elevatorDriveNotOk :=
        hmiAlarms.elevatorDriveNotOk OR
        NOT elevatorDriveOk;

    hmiAlarms.elevatorFault :=
        hmiAlarms.elevatorFault OR
        elevatorFault;

    hmiAlarms.elevatorNotHomed :=
        hmiAlarms.elevatorNotHomed OR
        (
            elevatorAutoCmd AND
            NOT elevatorHomed
        );

//    hmiAlarms.elevatorNotInPosition :=
//        hmiAlarms.elevatorNotInPosition OR
//        (
//            systemRunEnable AND
//            elevatorAutoCmd AND
//            elevatorHomed AND
//            NOT elevatorInPosition
//        );

    hmiAlarms.elevatorUpperSafetyLimitActive :=
        hmiAlarms.elevatorUpperSafetyLimitActive OR
        elevatorUpperSafetyLimit;

    hmiAlarms.elevatorLowerSafetyLimitActive :=
        hmiAlarms.elevatorLowerSafetyLimitActive OR
        elevatorLowerSafetyLimit;

    (*
    hmiAlarms.elevatorUpperLimitActive :=
        hmiAlarms.elevatorUpperLimitActive OR
        elevatorUpperLimit;

    hmiAlarms.elevatorLowerLimitActive :=
        hmiAlarms.elevatorLowerLimitActive OR
        elevatorLowerLimit;
    *)

END_IF;
END_METHOD

//==============================================================
// COMPLEX STACKER — BACKSTOP CONTROL
// EN: Controls the backstop axis with homing, manual movement,
//     automatic positioning, override positioning and protections.
//
// Signed speed convention:
// Positive = open
// Negative = close
//
// State code:
// 0  = STOP
// 10 = HOME_FAST_SEARCH
// 11 = HOME_SLOW_EXIT_SENSOR
// 12 = HOME_SET_ENCODER
// 13 = HOME_WAIT_AFTER_SET
// 14 = HOME_MOVE_TO_TARGET
// 20 = MANUAL
// 30 = AUTO_POSITION
// 40 = FAULT
//==============================================================
METHOD _BackstopControl



//==============================================================
// 1) Default internal commands
//==============================================================
// EN: Internal signed speed is reset every scan and set by the active state.
//     Positive = open, negative = close.
backstopSignedSpeedRefMmps := 0.0;

// EN: Internal trigger for encoder set pulse.
backstopSetEncoderPositionTrigger := FALSE;


//==============================================================
// 2) Edge detection
//==============================================================
// EN: Home can be requested manually by HMI or automatically by _SystemControl.
//     Automatic home is accepted only when backstopAutoCmd is enabled.
//     Movement is allowed only when master system run is enabled.
backstopHomeRequestCombined :=
    systemRunEnable AND
    (
        backstopHomeCmd OR
        (
            backstopAutoCmd AND
            backstopAutoHomeRequest
        )
    );

rBackstopHome :=
    backstopHomeRequestCombined AND
    NOT backstopHomeRequestCombinedOld;

backstopHomeRequestCombinedOld :=
    backstopHomeRequestCombined;


// EN: Execute positioning command edge.
//     This command only generates movement when system is enabled and backstop auto is enabled.
rBackstopExecutePositioning :=
    systemRunEnable AND
    backstopExecutePositioningCmd AND
    NOT backstopExecutePositioningCmdOld;

backstopExecutePositioningCmdOld := backstopExecutePositioningCmd;


// EN: Override falling edge.
//     Used as fallback to return to programmed position if override is released.
backstopTargetOverrideFallingEdge :=
    backstopTargetOverrideOld AND NOT backstopTargetOverrideActive;

backstopTargetOverrideOld := backstopTargetOverrideActive;


//==============================================================
// 3) Home limit selection and edge detection
//==============================================================
// EN: Home limit depends on configured homing direction.
IF machineConfig.backstopHomeDirection > 0 THEN

    backstopHomeLimitReached := backstopMaxLimit;

ELSIF machineConfig.backstopHomeDirection < 0 THEN

    backstopHomeLimitReached := backstopMinLimit;

ELSE

    backstopHomeLimitReached := FALSE;

END_IF;


// EN: Falling edge is used after the home limit has been reached.
backstopHomeLimitFallingEdge :=
    backstopHomeLimitOld AND NOT backstopHomeLimitReached;

backstopHomeLimitOld := backstopHomeLimitReached;


//==============================================================
// 4) Movement permissions
//==============================================================
backstopOpenAllowed :=
    systemRunEnable AND
    safetyCircuitOk AND
    backstopDriveOk AND
    NOT backstopMaxLimit AND
    NOT backstopSafeMaxLimit AND
    (
        (NOT backstopHomed) OR
        (backstopPositionMm < machineConfig.backstopMaxPositionMm)
    );

backstopCloseAllowed :=
    systemRunEnable AND
    safetyCircuitOk AND
    backstopDriveOk AND
    NOT backstopMinLimit AND
    NOT backstopSafeMinLimit AND
    (
        (NOT backstopHomed) OR
        (backstopPositionMm > machineConfig.backstopMinPositionMm)
    );


// EN: During homing, the normal home limit is allowed.
//     Only the safe limit blocks movement.
IF machineConfig.backstopHomeDirection > 0 THEN

    backstopHomeMoveAllowed :=
        systemRunEnable AND
        safetyCircuitOk AND
        backstopDriveOk AND
        NOT backstopSafeMaxLimit;

ELSIF machineConfig.backstopHomeDirection < 0 THEN

    backstopHomeMoveAllowed :=
        systemRunEnable AND
        safetyCircuitOk AND
        backstopDriveOk AND
        NOT backstopSafeMinLimit;

ELSE

    backstopHomeMoveAllowed := FALSE;

END_IF;


//==============================================================
// 5) Programmed / override target calculation
//==============================================================
// EN: Programmed target follows sheet length plus mechanical offset.
//     This value can change, but it does not move the backstop by itself.
backstopProgrammedTargetPositionMm :=
    LIMIT(
        machineConfig.backstopMinPositionMm,
        MAX(0.0, sheetLengthMm) + machineConfig.backstopSheetLengthOffsetMm,
        machineConfig.backstopMaxPositionMm
    );


// EN: Before homing, keep the latched target updated with programmed target.
//     This avoids an invalid old target after power-up.
IF NOT backstopHomed THEN

    backstopLatchedTargetPositionMm := backstopProgrammedTargetPositionMm;

END_IF;


//==============================================================
// 5.1) Automatic positioning request handling
//==============================================================
// EN: Auto mode only enables positioning. It does not execute positioning.
//     Normal positioning must be requested by backstopExecutePositioningCmd.
//     Override positioning is requested by the automatic cycle.
IF NOT systemRunEnable THEN

    backstopPositioningRequestActive := FALSE;


ELSIF NOT backstopAutoCmd THEN

    backstopPositioningRequestActive := FALSE;


ELSIF backstopTargetOverrideActive THEN

    // EN: Override has priority. Clear normal positioning request.
    backstopPositioningRequestActive := FALSE;


ELSIF rBackstopExecutePositioning THEN

    // EN: Latch current programmed target only when execute command is received.
    backstopLatchedTargetPositionMm := backstopProgrammedTargetPositionMm;
    backstopPositioningRequestActive := TRUE;


ELSIF backstopTargetOverrideFallingEdge THEN

